FUNCTION_BLOCK FB_ModePos
VAR_INPUT
	bExecute:BOOL;
	bReset: BOOL;
	fVelSet:LREAL:=0;
	fPosSet:LREAL:=0;
	stStatus: ST_AXIS_STATUS;
END_VAR
VAR_OUTPUT
	bError: BOOL;
	nErrorId: UDINT;
	sErrorStr: STRING:=GVL_ErrorCodes.nErrorCodeOKStr;
END_VAR
VAR_IN_OUT
	stCommands: ST_AXIS_COMMAND;
END_VAR
VAR

END_VAR

// Function: Absolute positioning of target main  motor
// Actual positioning will be performed by the drive.
// Author: Anders Sandström 2018

stCommands.eMotionMode :=e_Motion_mode.ePositioning;
stCommands.eOperationMode:=e_Operation_mode_no.eSecondaryOpMode1;
IF bExecute THEN
  stCommands.fVelocityCommandValue:=fVelSet;
ELSE
  stCommands.fVelocityCommandValue:=0;
END_IF
stCommands.fCommandVelocity:=0;
stCommands.fCommandPosition:=fPosSet;

END_FUNCTION_BLOCK

(* stored: Version 1.1.0.1, ProductVersion 3.1.4024.0
   POU FB_ModePos: Id {6ecfe6fb-3b6b-4228-bef4-e3d81387d91d}, SpecialFunc None *)
